// TIA Portal V20 export
TYPE "LConSMC_typeBreakPointTable"
// stored: Access Published
   STRUCT
      values : Array[0.."LCON_MAX_VALUE_BREAK_POINT_TABLE"] of LReal;
   END_STRUCT;
   // values[0..19] := 0.0;
END_TYPE
